FUNCTION_BLOCK Test_AssertEquals_STRING EXTENDS TUnitTestBase
VAR
    AssertionUnderTest : TAssertion(AssertionListenerMock);
    AssertionListenerMock : TAssertionListenerMock;
    STRING_Variable : STRING := 'Cucumber';
END_VAR

AssertionListenerMock.AssertionFailed  := FALSE;
AssertionListenerMock.AssertionMessage := '';
AssertionListenerMock.ExpectedAsString := '';
AssertionListenerMock.ActualAsString   := '';

// Test the assertion...
AssertionUnderTest.AssertEquals_STRING(
    Expected := 'Radish',
    Actual   := STRING_Variable,
    VariableName := 'STRING_Variable'); 
    
// Check the assertion worked...    
Assertion.AssertEquals_BOOL(
    Expected := TRUE,
    Actual   := AssertionListenerMock.AssertionFailed,
    VariableName := 'AssertionListenerMock.AssertionFailed');

// Check the assertion messages...    
Assertion.AssertEquals_STRING(
    Expected := 'AssertEquals_STRING failed in AssertionTest: Value "STRING_Variable"',
    Actual   := AssertionListenerMock.AssertionMessage,
    VariableName := 'AssertionListenerMock.AssertionMessage');

Assertion.AssertEquals_STRING(
    Expected := '  Expected = Radish',
    Actual   := AssertionListenerMock.ExpectedAsString,
    VariableName := 'AssertionListenerMock.ExpectedAsString');

Assertion.AssertEquals_STRING(
    Expected := '  Actual   = Cucumber',
    Actual   := AssertionListenerMock.ActualAsString,
    VariableName := 'AssertionListenerMock.ActualAsString');

TestFinished();

END_FUNCTION_BLOCK

(* stored: Version 1.1.0.1, ProductVersion 3.1.4024.4
   POU Test_AssertEquals_STRING: Id {28a1ba85-4d0f-431d-92ea-6bc505340d93}, SpecialFunc None *)
